TYPE ST_PSU_Inputs :
STRUCT
	bWarning 				: BOOL;
	bError 					: BOOL;
	bI2TWarning 			: BOOL;
	DCOk					: BOOL;
	Overrange				: BOOL;
	nInpuCycleCounter 		: UINT;
	fActualOutputVoltage 	: REAL;
	fActualOutputCurrent 	: REAL;
	nActualI2TUtilization 	: USINT;
	nInfoData1 				: UINT;
	nInfoData2 				: UINT;
END_STRUCT
END_TYPE

(* stored: Version 1.1.0.1
   DUT ST_PSU_Inputs: Id {304e99c6-5c53-4cc4-ac2f-ecad528ae4b3} *)
